INTERFACE I_Statehandler

METHOD SetState : BOOL
VAR_INPUT
	eNewState: E_STATES;
END_VAR
END_METHOD

END_INTERFACE

(* stored: Version 1.1.0.1, ProductVersion 3.1.4024.3
   Itf I_Statehandler: Id {6ad18ada-1fb5-48cb-8dc1-c2679983afa6}
   Method SetState: Id {fefb3d48-6184-40f2-9ec0-ad0740b0c9d9} *)
